Yaskawa INFORM job: MAT.JBI

/JOB
//NAME MAT
//POS
///NPOS 3,0,0,0
///TOOL 0
///PULSE
C000=-28576,31503,-16829,3172,10081,-9916
C001=-28765,32157,-17684,2578,10064,9824
C002=-28793,32127,-17637,2615,10057,-7799
//INST
///DATE 2014/10/11 22:58
///ATTR 0,0,0,0,0,0,0,0,0,0,0,0,0,1,0,0
///FRAME BASE
NOP
*1
MOVJ C000 VJ=100.00 CONT
MOVJ C001 VJ=100.00 CONT
MOVJ C002 VJ=100.00 CONT
JUMP *1
END
